{attribute 'GeneratedUsingTerminal: IL2302-B110-0016'}
{attribute addProperty BoxType "IL2302-B110-0016"}
{attribute addProperty Id "InputsAT %I*Inputs_CC16D1F40OutputsAT %I*Outputs_D8BAB3B30WcStateAT %I*WcState_9091E0EB2InfoDataAT %I*InfoData_41C547A32"}
{attribute addProperty CRC "323002079"}
{attribute addProperty Size "4"}
TYPE IL2302_13409EDF EXTENDS EtcSlaveTerminalBase_947E5A46 :
STRUCT
	{attribute addProperty Name "Inputs"}
	Inputs : Inputs_CC16D1F4;
	{attribute addProperty Name "Outputs"}
	Outputs : Outputs_D8BAB3B3;
	{attribute addProperty Name "WcState"}
	WcState : WcState_9091E0EB;
	{attribute addProperty Name "InfoData"}
	InfoData : InfoData_41C547A3;
END_STRUCT
END_TYPE

(* stored: Version 1.2.0.0, ProductVersion 3.1.4024.9
   DUT IL2302_13409EDF: Id {a3d53661-91a2-4244-94ab-c6c80d519744} *)
